{attribute 'GeneratedUsingTerminal: EPP9001-0060-0016'}
{attribute addProperty BoxType "EPP9001-0060-0016"}
{attribute addProperty Id "InfoDataAT %I*InfoData_6F19DB2B2"}
{attribute addProperty CRC "532711307"}
{attribute addProperty Size "2"}
TYPE EPP9001_1FC0878B EXTENDS EtcSlaveTerminalBase_947E5A46 :
STRUCT
	{attribute addProperty Name "InfoData"}
	InfoData : InfoData_6F19DB2B;
END_STRUCT
END_TYPE

(* stored: Version 1.2.0.0, ProductVersion 3.1.4024.9
   DUT EPP9001_1FC0878B: Id {341b5fa0-1f64-45bf-9dd9-43abe19c0961} *)
